// TIA Portal V19 export
TYPE "lexchangetray_typeplasticWorkStation_signalTM_Monitor"
// Type: Bool
// stored: Access Published
   STRUCT
      simulationed : Bool;
      inspectionAfterPlasticTrayJacking : Bool;   // 塑胶顶升后检测
      inspectionBeforePlasticTrayJacking : Bool;   // 塑胶顶升前检测
      plasticTrayFeedingDetection : Bool;   // 塑胶托盘入料检测
      plasticTrayLiftingCylinderHomePositionDetection1 : Bool;   // 塑胶顶升气缸1原位检测
      plasticTrayTrayInplaceDetection : Bool;   // 塑胶托盘到位检测
      plasticTrayLiftingCylinderWorkingPositionDetection1 : Bool;   // 塑胶顶升气缸1工作位检测
      scapegoatSignal1 : Bool;   // 替罪羊1信号
      scapegoatSignal2 : Bool;   // 替罪羊2信号
   END_STRUCT;
END_TYPE
